Fanuc KAREL source: kt00485.KL

-- PROVISIONAL review KL for V770-1; original PC SHA256 b852c1b72b94e707e976269951cd582077acedbb5dafe9745467098ae0288601
-- Incomplete behavior may be omitted. Consult companion uncertainty JSON. Do not deploy.
PROGRAM KT00485
%NOLOCKGROUP
-- UNRESOLVED_DECL P1 type=000101
-- UNRESOLVED_DECL P2 type=000106
-- UNRESOLVED_DECL OUT type=000102
BEGIN
  -- UNRESOLVED_PC offsets 5-20; opcodes 2E,22,32,35
  -- UNRESOLVED_PC offsets 25-59; opcodes 49,49,7E,60,7E,4A
  -- UNRESOLVED_PC offsets 64-68; opcodes 7F
END KT00485
